{attribute 'qualified_only'}
VAR_GLOBAL
	nn : Layers;
END_VAR

(* stored: Version 1.1.0.1, ProductVersion 3.1.4024.12
   GVL GVL_NN: Id {450fdbfe-f218-4ffe-938f-15bed2b64745} *)
